# EPICS substitutions: RFMonitor/rfMonitorApp/Db/userHost.substitutions
# Example substitutions file

file "db/dbExample1.db" {
    { user = "longHost" }
}

file db/dbExample2.db {
    pattern { user, no, scan }
        { "longHost", 1, "1 second" }
        { "longHost", 2, "2 second" }
        { "longHost", 3, "5 second" }
}
